// TIA Portal V17 export
// export: Created 2025-06-26T06:49:26.7197768Z, ExportSetting WithDefaults, DisplayName Totally Integrated Automation Portal, DisplayVersion V17 Update 8, DisplayName TIA Portal Openness, DisplayVersion V17 Update 8, DisplayName TIA Portal Version Control Interface, DisplayVersion V17, DisplayName STEP 7 Professional, DisplayVersion V17 Update 8, DisplayName STEP 7 Safety, DisplayVersion V17 Update 6, DisplayName WinCC Advanced, DisplayVersion V17 Update 8
TYPE "stRawValue"
// stored: IsFailsafeCompliant false
   STRUCT
      iMin : Int;   // Module output at minimum input
      iMax : Int;   // Module output at maximum input
      iValue : Int;   // Current module value
      bFault : Bool;   // 0 = valid data, 1 = invalid data
   END_STRUCT;
END_TYPE
